// TIA Portal V18 export
TYPE "UDT_ACsDO"
// stored: IsFailsafeCompliant false
   STRUCT
      xACCentralEnable : Bool;
   END_STRUCT;
END_TYPE
